FUNCTION_BLOCK IA_VDS (* ISOBUS Adapter for Vehicle Direction/Speed (VDS) *)
  (* Standard: ISO 11783-7; Classification: PGN 65256; Description: Copyright (c) 2024-2026 HR Agrartechnik GmbH This program and the accompanying materials are made available under the terms of the Eclipse Public License 2.0 which is available at https://www.eclipse.org/legal/epl-2.0/ SPDX-License-Identifier: EPL-2.0 *)
  (* Version 1.3, 2026-09-17, Franz Höpfinger, HR Agrartechnik GmbH, Dokumentation (Franz: 'das passt, wir dokumentieren das in den Bausteinen. E_D_FF ist ein IEC 61499 Standardbaustein, wir halten uns STRENG an die Norm. E_D_FF_ANY ist davon abgeleitet, sollte sich gleich verhalten'): E_D_FF_Timeout (E_D_FF, IEC 61499-1 Annex A Standardbaustein) feuert EO NICHT beim allerersten CLK, wenn der erste echte Wert mit dem default-initialisierten Vergleichszustand (FALSE) uebereinstimmt - bleibt I_VDS.Q_timeout von Anfang an FALSE (Normalfall, kein Timeout), feuert TIMEOUT.E1 nie initial. Bewusst kein Bug, sondern standardkonformes Verhalten (analog E_RS/E_SR, wo genau dasselbe Verhalten Anlass fuer die Sonderformen E_RS_SYM/E_SR_SYM war) - hier bewusst KEINE eigene SYM-Variante, da nachgelagerte Verbraucher TIMEOUT.D1 als Datenwert lesen, nicht nur das Event. *)
  (* Version 1.2, 2026-09-17, Franz Höpfinger, HR Agrartechnik GmbH, Bugfix (PR #241 Review, qodo-code-review[bot]: 'Normal traffic floods timeout consumers - every IND republishes Q_timeout even when it did not change'): E_D_FF_Timeout (E_D_FF_ANY) vor TIMEOUT eingefuegt, wie schon fuer die anderen Signale dieser Datei - I_VDS.TIMEOUT und I_VDS.IND feuern jetzt beide nur noch E_D_FF_Timeout.CLK, TIMEOUT.E1/D1 werden nur noch bei tatsaechlicher Aenderung von Q_timeout aktualisiert, nicht mehr bei jeder einzelnen Botschaft im gesunden Normalbetrieb. *)
  (* Version 1.1, 2026-09-16, Franz Höpfinger, HR Agrartechnik GmbH, E_D_FF_ANY-Aenderungsfilter fuer NAV_SPEED/BEARING/ALTITUDE ergaenzt (analog IA_RPTO v1.1). *)
  PACKAGE isobus::tecu;
  (* Documentation:
  ISOBUS Adapter for Vehicle Direction/Speed (VDS)
   TIMEOUT.E1-Verdrahtung: I_VDS.TIMEOUT (echter Timeout-Eintritt) UND I_VDS.IND (Normalbetrieb) feuern beide E_D_FF_Timeout.CLK; E_D_FF_Timeout (E_D_FF_ANY, gespeist von I_VDS.Q_timeout) laesst TIMEOUT.E1 nur bei tatsaechlicher Wertaenderung durch - so wird TIMEOUT.D1 (Q_timeout) am Adapter-Plug beim Zuruecksetzen auf false weiterhin zuverlaessig aktualisiert, ohne bei jeder einzelnen Botschaft im gesunden Normalbetrieb erneut zu feuern. Der zugrundeliegende TIMEOUT/IND-Vertrag von I_VDS selbst ist in dessen eigener .fbt-Datei dokumentiert.
  *)
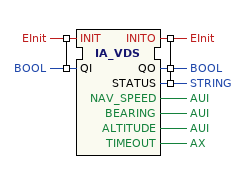
  EVENT_INPUT
    INIT : EInit WITH QI; (* Service Initialization *)
  END_EVENT
  EVENT_OUTPUT
    INITO : EInit WITH QO, STATUS; (* Initialization Confirm *)
  END_EVENT
  VAR_INPUT
    QI : BOOL; (* Event Input Qualifier *)
  END_VAR
  VAR_OUTPUT
    QO : BOOL; (* Event Output Qualifier *)
    STATUS : STRING;
  END_VAR
  PLUGS
    NAV_SPEED : adapter::types::unidirectional::AUI; (* Navigation-based vehicle speed *)
    BEARING : adapter::types::unidirectional::AUI; (* Compass bearing *)
    ALTITUDE : adapter::types::unidirectional::AUI; (* Altitude *)
    TIMEOUT : adapter::types::unidirectional::AX; (* Timeout Status *)
  END_PLUGS
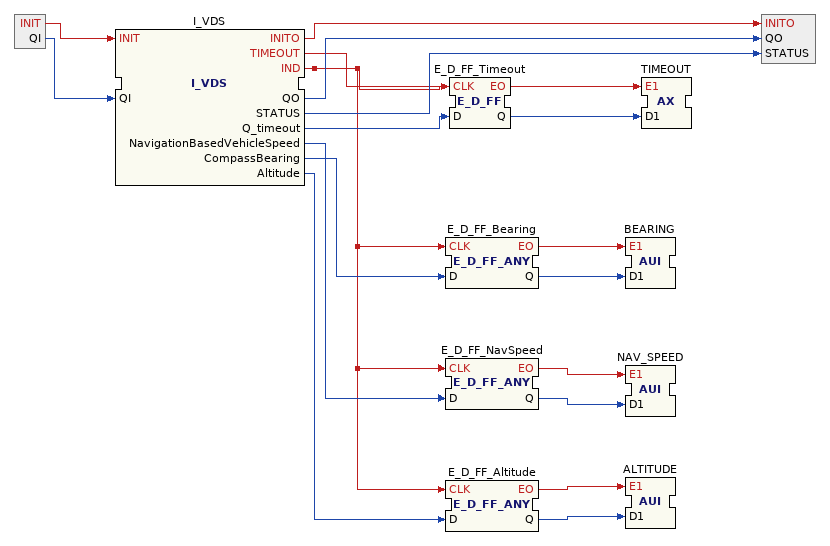
  FBS
    I_VDS : isobus::tecu::I_VDS;
    E_D_FF_NavSpeed : iec61499::events::E_D_FF_ANY;
    E_D_FF_Bearing : iec61499::events::E_D_FF_ANY;
    E_D_FF_Altitude : iec61499::events::E_D_FF_ANY;
    E_D_FF_Timeout : iec61499::events::E_D_FF;
  END_FBS
  EVENT_CONNECTIONS
    INIT TO I_VDS.INIT;
    I_VDS.INITO TO INITO;
    I_VDS.TIMEOUT TO E_D_FF_Timeout.CLK;
    I_VDS.IND TO E_D_FF_NavSpeed.CLK;
    E_D_FF_NavSpeed.EO TO NAV_SPEED.E1;
    I_VDS.IND TO E_D_FF_Bearing.CLK;
    E_D_FF_Bearing.EO TO BEARING.E1;
    I_VDS.IND TO E_D_FF_Altitude.CLK;
    E_D_FF_Altitude.EO TO ALTITUDE.E1;
    I_VDS.IND TO E_D_FF_Timeout.CLK;
    E_D_FF_Timeout.EO TO TIMEOUT.E1;
  END_CONNECTIONS
  DATA_CONNECTIONS
    QI TO I_VDS.QI;
    I_VDS.QO TO QO;
    I_VDS.STATUS TO STATUS;
    I_VDS.Q_timeout TO E_D_FF_Timeout.D;
    E_D_FF_Timeout.Q TO TIMEOUT.D1;
    I_VDS.NavigationBasedVehicleSpeed TO E_D_FF_NavSpeed.D;
    E_D_FF_NavSpeed.Q TO NAV_SPEED.D1;
    I_VDS.CompassBearing TO E_D_FF_Bearing.D;
    E_D_FF_Bearing.Q TO BEARING.D1;
    I_VDS.Altitude TO E_D_FF_Altitude.D;
    E_D_FF_Altitude.Q TO ALTITUDE.D1;
  END_CONNECTIONS
END_FUNCTION_BLOCK
